FUNCTION F_DerotatorPosition2 : LREAL
VAR_INPUT
	// azimuth of the target
	azimuth: LREAL;
	// elevation of the target in degrees
	elevation: LREAL;
	// declination of the target in degrees
	declination: LREAL;
	// latitude in degrees
	latitude:	LREAL;
	// sign for elevation
	sign:	LREAL := 1.0;
END_VAR
VAR
	// parallactic angle
	de, az, el, la: LREAL;
	parallactic_angle:	LREAL;
	//zenith_distance: LREAL;
END_VAR
VAR CONSTANT
	d2r:	LREAL := PI/180.0;
	r2d:	LREAL := 180.0/PI;
	//h2r:	LREAL := PI/12.0;
	//h2d:	LREAL := 15.0;
END_VAR

// calculate the parallactic angle
de := LIMIT(-90.0, declination, 90.0) * d2r;
az := MODABS(azimuth, 360.0) * d2r;
el := LIMIT(0.0, elevation, 90.0) * d2r;
la := LIMIT(-90.0, latitude, 90.0) * d2r;

parallactic_angle := - r2d * ATAN2(SIN(az), TAN(la)*COS(el)-SIN(el)*COS(az));

F_DerotatorPosition2 := parallactic_angle - sign * elevation;
F_DerotatorPosition2 := MODABS(F_DerotatorPosition2, 360.0);

END_FUNCTION

(* stored: Version 1.1.0.1, ProductVersion 3.1.4024.12
   POU F_DerotatorPosition2: Id {e646c6f5-cf02-4188-95c2-c7b920ede3a4}, SpecialFunc None *)
